// TIA Portal V20 export
TYPE "HMI_VlvMotL"
   STRUCT
      OpenMan : Bool := FALSE;   // 1=Open: Open Command in Manual Mode
      CloseMan : Bool := FALSE;   // 1=Close: Close Command in Manual Mode
      StopMan : Bool := FALSE;   // 1=Stop: Stop Command in Manual Mode
      AutModOp : Bool := FALSE;   // 1=Auto Mode: Auto Mode by Operator
      ManModOp : Bool := TRUE;   // 1=Manual Mode: Manual Mode by Operator
      LocalLi : Bool;   // 1=Local Mode: Local Operation by Field Signal
      LocalOp : Bool := FALSE;   // 1=Local Mode: Local Operation by Operator
      OosOp : Bool := FALSE;   // 1=Oos Mode: Oos Mode by Operator
      OpenLocal : Bool;   // 1=Start Local: Field Open Signal
      CloseLocal : Bool;   // 1=Start Local: Field Close Signal
      StopLocal : Bool;   // 1=Stop Local: Field Stop Signal
      V_Monitor : Bool := TRUE;   // 1=Monitor ON, 0=Monitor OFF: Valve Feedback Monitor
      V_MonTiStatic : Real := 5.0;   // Valve Monitoring Time of Feedback [s]
      V_MonTiDynamic : Real := 5.0;   // Valve Monitoring Time of Feedback [s]
      M_Monitor : Bool := TRUE;   // 1=Monitor ON, 0=Monitor OFF: Motor Feedback Monitor
      M_MonTiStatic : Real := 3.0;   // Motor Monitoring Time of Feedback [s]
      M_MonTiDynamic : Real := 3.0;   // Motor Monitoring Time of Feedback on starting or on change in control output [s
      M_MonTiStop : Real := 3.0;   // Motor Monitoring Time of Feedback on stopping in control output [s]
      RapidStp : Bool := FALSE;   // 1 = Motor Rapid Stop command
      RstOp : Bool := FALSE;   // Operator Reset Signal
      BypProt : Bool := FALSE;   // Bypass Protection in Sim/Local Modes
      Permit_ST : Byte := BYTE#16#FF;   // Permit Signal Status
      PermCls_ST : Byte := BYTE#16#FF;   // PermCls Signal Status
      Intlock_ST : Byte := BYTE#16#FF;   // Intlock Signal Status
      IntlCls_ST : Byte := BYTE#16#FF;   // IntlCls Signal Status
      Protect_ST : Byte := BYTE#16#FF;   // Protect Signal Status
      ProtCls_ST : Byte := BYTE#16#FF;   // ProtCls Signal Status
      TorqOpen : Bool := true;   // 1=Normal, 0=Torque Open is High
      TorqClose : Bool := true;   // 1=Normal, 0=Torque Close is High
      UserAna1 : Real;   // User Analog Input 1
      UA1unit : Int := 0;   // Unit of UserAna1
      UserAna2 : Real;   // User Analog Input 2
      UA2unit : Int := 0;   // Unit of UserAna2
      BatchID : DWord := 16#0;   // Current Batch ID (number)
      BatchName : String[32] := '';   // Current Batch Name
      StepNo : DWord := 16#0;   // Batch Step Number
      CurrMonV { ExternalWritable := 'False'} : DInt := 0;   // Remaining monitoring time of valve [s]
      CurrMonM { ExternalWritable := 'False'} : DInt := 0;   // Remaining monitoring time of motor [s]
      FbkOpenOut { ExternalWritable := 'False'} : Bool;   // 1=Open : Feedback of Control Open
      FbkCloseOut { ExternalWritable := 'False'} : Bool;   // 1=Close : Feedback of Control Close
      FbkOpngOut { ExternalWritable := 'False'} : Bool;   // 1=Opening, 0=Stop: Feedback of Control Open
      FbkClsgOut { ExternalWritable := 'False'} : Bool;   // 1=Closing, 0=Stop: Feedback of Control Close
      OS_PermOut { ExternalWritable := 'False'} : DWord := DWORD#16#FFFF_FFFF;   // Operator Permission: Output for OS
      OS_PermLog { ExternalWritable := 'False'} : DWord := DWORD#16#FFFF_FFFF;   // Operator Permission: Output for OS
      OpSt_Out { ExternalWritable := 'False'} : DWord := 16#0;   // Enabled operator stations
      ST_Worst { ExternalWritable := 'False'} : Byte := 16#80;   // Worst Signal Status
      AutoST { ExternalWritable := 'False'} : Byte := 16#80;   // Worst Signal Status of the automatic commands
      Status1 { ExternalWritable := 'False'} : DWord := 16#0;   // Status1 Word
      Status2 { ExternalWritable := 'False'} : DWord := 16#0;   // Status2 Word
      Status3 { ExternalWritable := 'False'} : DWord := 16#0;   // Status3 Word
      Status4 { ExternalWritable := 'False'} : DWord := 16#0;   // Status4 Word
      Status5 { ExternalWritable := 'False'} : DWord := 16#0;   // Status5 Word
      AlarmState { ExternalWritable := 'False'} : Word;   // Alarm State for group display / Alarm Status for group display
   END_STRUCT;
END_TYPE
